PROGRAM MOTOR_FAULTS
VAR
	TON_GL1_MTR: TON; // MOTOR FAULT DELAY TIMER
	TON_GL2_MTR: TON; // MOTOR FAULT DELAY TIMER
	TON_GL3_MTR: TON; // MOTOR FAULT DELAY TIMER
	TON_GL4_MTR: TON; // MOTOR FAULT DELAY TIMER
	TON_GL5A_MTR: TON; // MOTOR FAULT DELAY TIMER
	TON_GL5B_MTR: TON; // MOTOR FAULT DELAY TIMER
	TON_GL6_MTR: TON; // MOTOR FAULT DELAY TIMER
	TON_GL7_MTR: TON; // MOTOR FAULT DELAY TIMER
	TON_GL8_MTR: TON; // MOTOR FAULT DELAY TIMER
	TON_GL9_MTR: TON; // MOTOR FAULT DELAY TIMER
	TON_GL10_MTR: TON; // MOTOR FAULT DELAY TIMER
	TON_GL11_MTR: TON; // MOTOR FAULT DELAY TIMER
	
	GL1_MTR: sClearPath;
	GL2_MTR: sClearPath;
	GL3_MTR: sClearPath;
	GL4_MTR: sClearPath;
	GL5_MTR: sClearPath;
	GL6_MTR: sClearPath;
	GL7_MTR: sClearPath;
	GL8_MTR: sClearPath;
	GL9_MTR: sClearPath;
	GL10_MTR: sClearPath;
	GL11_MTR: sClearPath;
		
	
	GL1: sTransfer;
	GL2: sTransfer;
	GL3: sConveyor;
	GL4: sConveyor;
	GL5A: sConveyor;
	GL5B: sConveyor;
	GL6: sConveyor;
	GL7:sConveyor;
	GL8: sConveyor;
	GL9: sConveyor;
	GL10: sConveyor;
	GL11: sConveyor;
	GL1_RD: SRoll_Door;
	

	RUN_FWD_TO_GL6_BIT : BOOL; // GL2 OCCUPIED, GL6 REQUESTING PART, RUN TO GL6 POSITION
	RUN_FWD_TO_GL8_BIT : BOOL; // GL2 OCCUPIED, GL8 REQUESTING PART, RUN TO GL8 POSITION
	RUN_REV_TO_GL5B_BIT : BOOL; //GL2 EMPTY, GL2 REQUESTING PART, RUN TO GL5 POSITION
	MTR_FAULT_PRESET_TIME: TIME; // FAULT TIMER PRESET TO MOTOR FAULT. DEFAULT IS 1000mS.
	COUNTER_PRESET: WORD; // MAX COUNT VALUE
	
	
END_VAR
VAR // added by the converter: edge detectors and wires of the graphical bodies
    _w1 : BOOL;
END_VAR

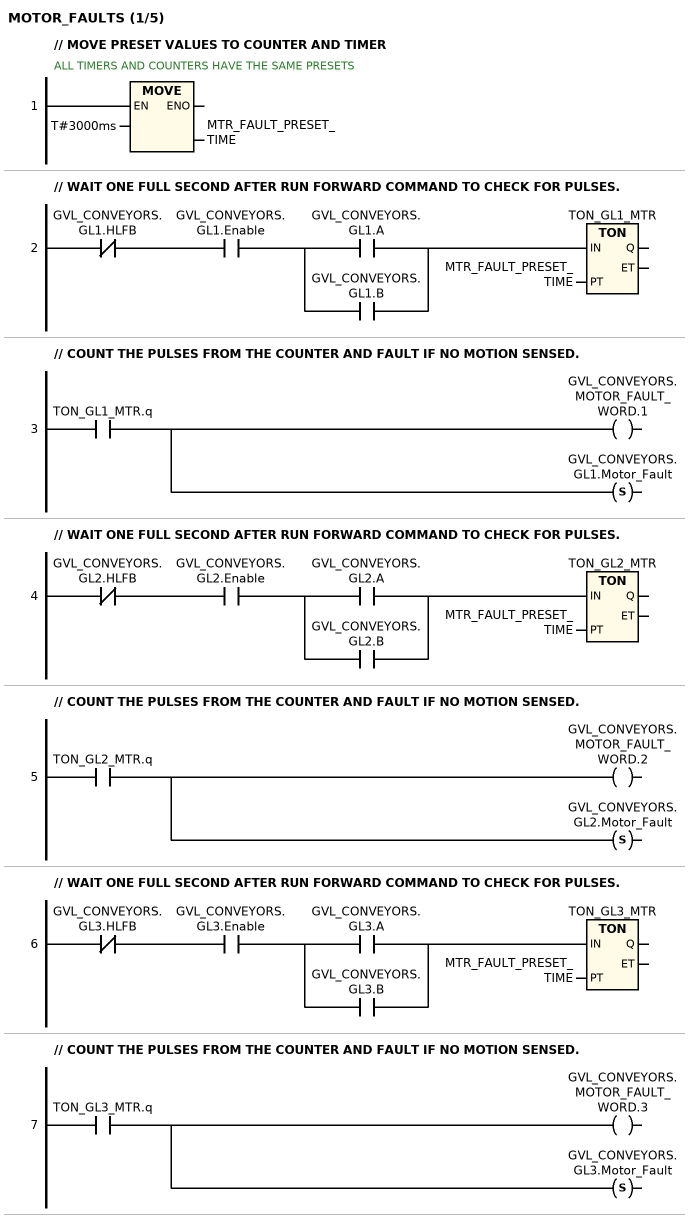
// NETWORK 1: // MOVE PRESET VALUES TO COUNTER AND TIMER
// ALL TIMERS AND COUNTERS HAVE THE SAME PRESETS
MTR_FAULT_PRESET_TIME := T#3000ms;

// NETWORK 2: // WAIT ONE FULL SECOND AFTER RUN FORWARD COMMAND TO CHECK FOR PULSES.
TON_GL1_MTR(IN := NOT GVL_CONVEYORS.GL1.HLFB AND GVL_CONVEYORS.GL1.Enable AND (GVL_CONVEYORS.GL1.A OR GVL_CONVEYORS.GL1.B), PT := MTR_FAULT_PRESET_TIME); // TON

// NETWORK 3: // COUNT THE PULSES FROM THE COUNTER AND FAULT IF NO MOTION SENSED.
GVL_CONVEYORS.MOTOR_FAULT_WORD.1 := TON_GL1_MTR.q;
GVL_CONVEYORS.GL1.Motor_Fault S= TON_GL1_MTR.q;

// NETWORK 4: // WAIT ONE FULL SECOND AFTER RUN FORWARD COMMAND TO CHECK FOR PULSES.
TON_GL2_MTR(IN := NOT GVL_CONVEYORS.GL2.HLFB AND GVL_CONVEYORS.GL2.Enable AND (GVL_CONVEYORS.GL2.A OR GVL_CONVEYORS.GL2.B), PT := MTR_FAULT_PRESET_TIME); // TON

// NETWORK 5: // COUNT THE PULSES FROM THE COUNTER AND FAULT IF NO MOTION SENSED.
GVL_CONVEYORS.MOTOR_FAULT_WORD.2 := TON_GL2_MTR.q;
GVL_CONVEYORS.GL2.Motor_Fault S= TON_GL2_MTR.q;

// NETWORK 6: // WAIT ONE FULL SECOND AFTER RUN FORWARD COMMAND TO CHECK FOR PULSES.
TON_GL3_MTR(IN := NOT GVL_CONVEYORS.GL3.HLFB AND GVL_CONVEYORS.GL3.Enable AND (GVL_CONVEYORS.GL3.A OR GVL_CONVEYORS.GL3.B), PT := MTR_FAULT_PRESET_TIME); // TON

// NETWORK 7: // COUNT THE PULSES FROM THE COUNTER AND FAULT IF NO MOTION SENSED.
GVL_CONVEYORS.MOTOR_FAULT_WORD.3 := TON_GL3_MTR.q;
GVL_CONVEYORS.GL3.Motor_Fault S= TON_GL3_MTR.q;

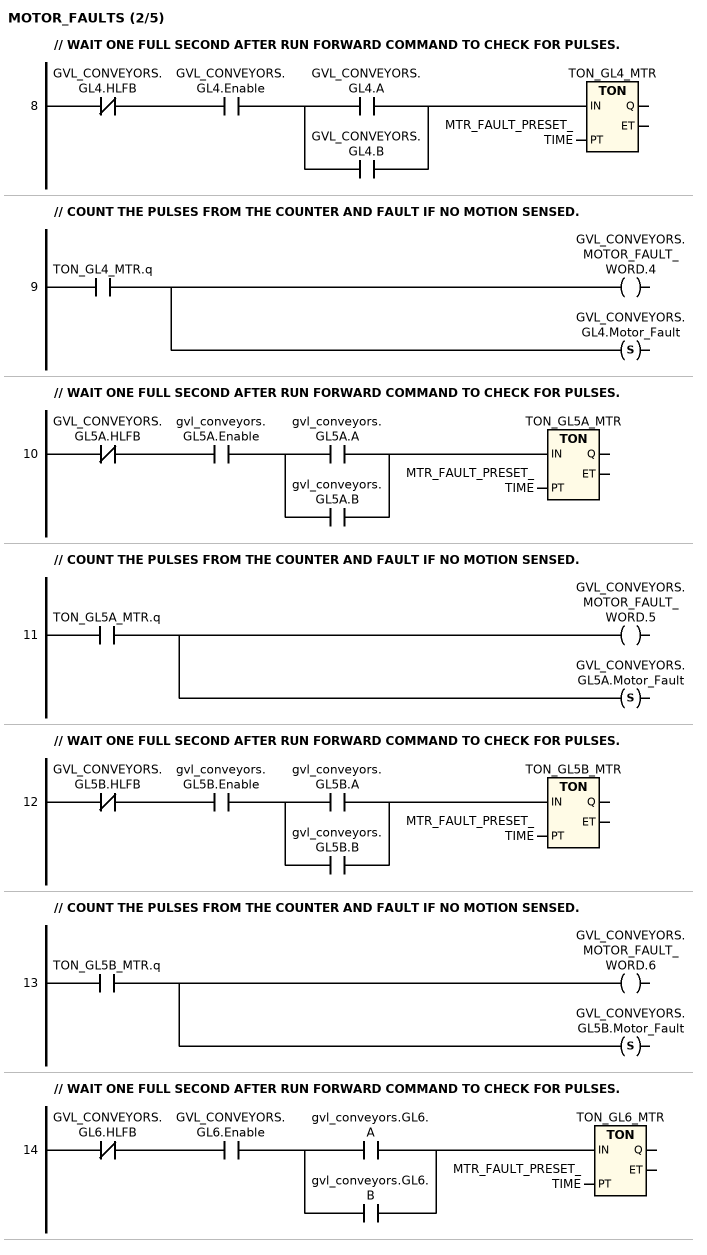
// NETWORK 8: // WAIT ONE FULL SECOND AFTER RUN FORWARD COMMAND TO CHECK FOR PULSES.
TON_GL4_MTR(IN := NOT GVL_CONVEYORS.GL4.HLFB AND GVL_CONVEYORS.GL4.Enable AND (GVL_CONVEYORS.GL4.A OR GVL_CONVEYORS.GL4.B), PT := MTR_FAULT_PRESET_TIME); // TON

// NETWORK 9: // COUNT THE PULSES FROM THE COUNTER AND FAULT IF NO MOTION SENSED.
GVL_CONVEYORS.MOTOR_FAULT_WORD.4 := TON_GL4_MTR.q;
GVL_CONVEYORS.GL4.Motor_Fault S= TON_GL4_MTR.q;

// NETWORK 10: // WAIT ONE FULL SECOND AFTER RUN FORWARD COMMAND TO CHECK FOR PULSES.
TON_GL5A_MTR(IN := NOT GVL_CONVEYORS.GL5A.HLFB AND gvl_conveyors.GL5A.Enable AND (gvl_conveyors.GL5A.A OR gvl_conveyors.GL5A.B), PT := MTR_FAULT_PRESET_TIME); // TON

// NETWORK 11: // COUNT THE PULSES FROM THE COUNTER AND FAULT IF NO MOTION SENSED.
GVL_CONVEYORS.MOTOR_FAULT_WORD.5 := TON_GL5A_MTR.q;
GVL_CONVEYORS.GL5A.Motor_Fault S= TON_GL5A_MTR.q;

// NETWORK 12: // WAIT ONE FULL SECOND AFTER RUN FORWARD COMMAND TO CHECK FOR PULSES.
TON_GL5B_MTR(IN := NOT GVL_CONVEYORS.GL5B.HLFB AND gvl_conveyors.GL5B.Enable AND (gvl_conveyors.GL5B.A OR gvl_conveyors.GL5B.B), PT := MTR_FAULT_PRESET_TIME); // TON

// NETWORK 13: // COUNT THE PULSES FROM THE COUNTER AND FAULT IF NO MOTION SENSED.
GVL_CONVEYORS.MOTOR_FAULT_WORD.6 := TON_GL5B_MTR.q;
GVL_CONVEYORS.GL5B.Motor_Fault S= TON_GL5B_MTR.q;

// NETWORK 14: // WAIT ONE FULL SECOND AFTER RUN FORWARD COMMAND TO CHECK FOR PULSES.
TON_GL6_MTR(IN := NOT GVL_CONVEYORS.GL6.HLFB AND GVL_CONVEYORS.GL6.Enable AND (gvl_conveyors.GL6.A OR gvl_conveyors.GL6.B), PT := MTR_FAULT_PRESET_TIME); // TON

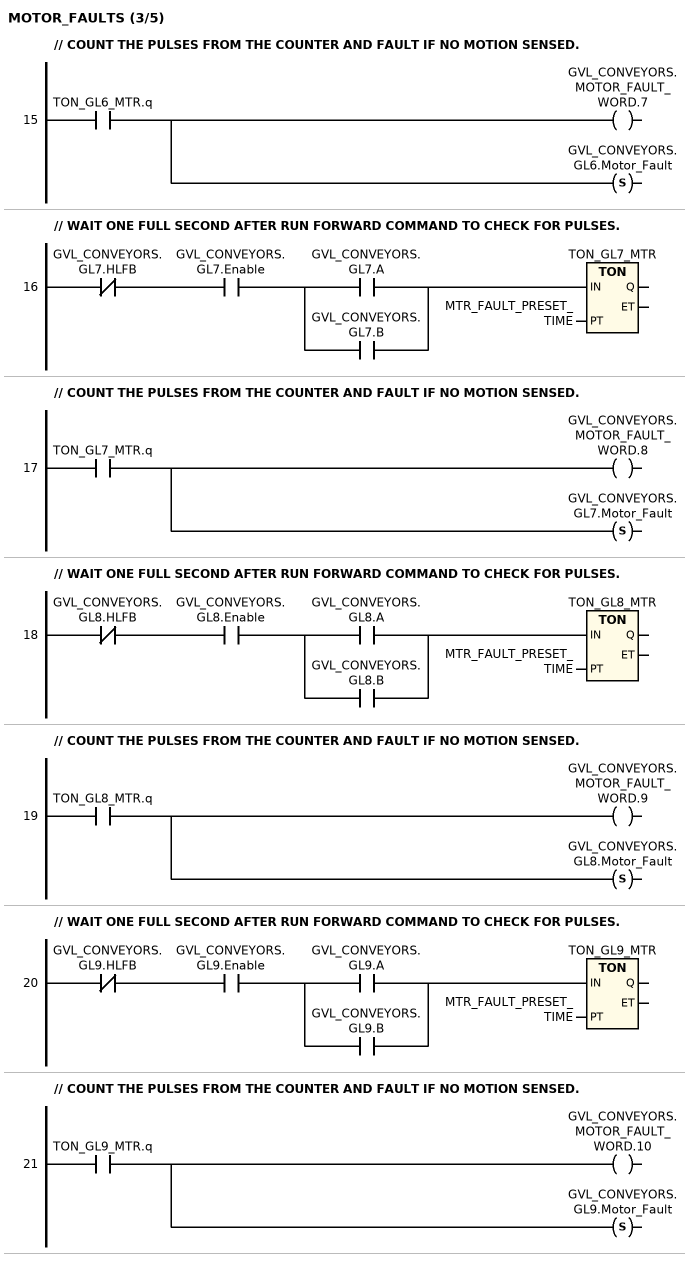
// NETWORK 15: // COUNT THE PULSES FROM THE COUNTER AND FAULT IF NO MOTION SENSED.
GVL_CONVEYORS.MOTOR_FAULT_WORD.7 := TON_GL6_MTR.q;
GVL_CONVEYORS.GL6.Motor_Fault S= TON_GL6_MTR.q;

// NETWORK 16: // WAIT ONE FULL SECOND AFTER RUN FORWARD COMMAND TO CHECK FOR PULSES.
TON_GL7_MTR(IN := NOT GVL_CONVEYORS.GL7.HLFB AND GVL_CONVEYORS.GL7.Enable AND (GVL_CONVEYORS.GL7.A OR GVL_CONVEYORS.GL7.B), PT := MTR_FAULT_PRESET_TIME); // TON

// NETWORK 17: // COUNT THE PULSES FROM THE COUNTER AND FAULT IF NO MOTION SENSED.
GVL_CONVEYORS.MOTOR_FAULT_WORD.8 := TON_GL7_MTR.q;
GVL_CONVEYORS.GL7.Motor_Fault S= TON_GL7_MTR.q;

// NETWORK 18: // WAIT ONE FULL SECOND AFTER RUN FORWARD COMMAND TO CHECK FOR PULSES.
TON_GL8_MTR(IN := NOT GVL_CONVEYORS.GL8.HLFB AND GVL_CONVEYORS.GL8.Enable AND (GVL_CONVEYORS.GL8.A OR GVL_CONVEYORS.GL8.B), PT := MTR_FAULT_PRESET_TIME); // TON

// NETWORK 19: // COUNT THE PULSES FROM THE COUNTER AND FAULT IF NO MOTION SENSED.
GVL_CONVEYORS.MOTOR_FAULT_WORD.9 := TON_GL8_MTR.q;
GVL_CONVEYORS.GL8.Motor_Fault S= TON_GL8_MTR.q;

// NETWORK 20: // WAIT ONE FULL SECOND AFTER RUN FORWARD COMMAND TO CHECK FOR PULSES.
TON_GL9_MTR(IN := NOT GVL_CONVEYORS.GL9.HLFB AND GVL_CONVEYORS.GL9.Enable AND (GVL_CONVEYORS.GL9.A OR GVL_CONVEYORS.GL9.B), PT := MTR_FAULT_PRESET_TIME); // TON

// NETWORK 21: // COUNT THE PULSES FROM THE COUNTER AND FAULT IF NO MOTION SENSED.
GVL_CONVEYORS.MOTOR_FAULT_WORD.10 := TON_GL9_MTR.q;
GVL_CONVEYORS.GL9.Motor_Fault S= TON_GL9_MTR.q;

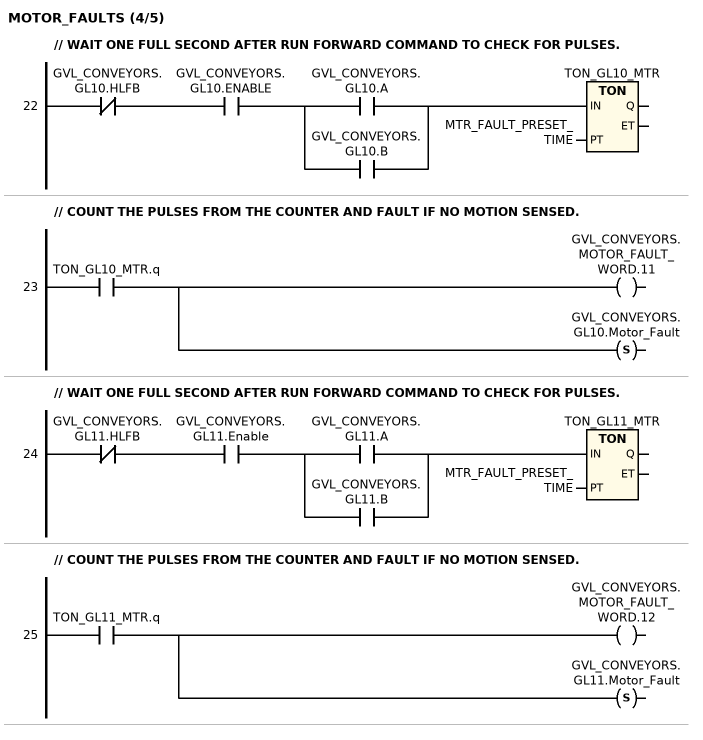
// NETWORK 22: // WAIT ONE FULL SECOND AFTER RUN FORWARD COMMAND TO CHECK FOR PULSES.
TON_GL10_MTR(IN := NOT GVL_CONVEYORS.GL10.HLFB AND GVL_CONVEYORS.GL10.ENABLE AND (GVL_CONVEYORS.GL10.A OR GVL_CONVEYORS.GL10.B), PT := MTR_FAULT_PRESET_TIME); // TON

// NETWORK 23: // COUNT THE PULSES FROM THE COUNTER AND FAULT IF NO MOTION SENSED.
GVL_CONVEYORS.MOTOR_FAULT_WORD.11 := TON_GL10_MTR.q;
GVL_CONVEYORS.GL10.Motor_Fault S= TON_GL10_MTR.q;

// NETWORK 24: // WAIT ONE FULL SECOND AFTER RUN FORWARD COMMAND TO CHECK FOR PULSES.
TON_GL11_MTR(IN := NOT GVL_CONVEYORS.GL11.HLFB AND GVL_CONVEYORS.GL11.Enable AND (GVL_CONVEYORS.GL11.A OR GVL_CONVEYORS.GL11.B), PT := MTR_FAULT_PRESET_TIME); // TON

// NETWORK 25: // COUNT THE PULSES FROM THE COUNTER AND FAULT IF NO MOTION SENSED.
GVL_CONVEYORS.MOTOR_FAULT_WORD.12 := TON_GL11_MTR.q;
GVL_CONVEYORS.GL11.Motor_Fault S= TON_GL11_MTR.q;

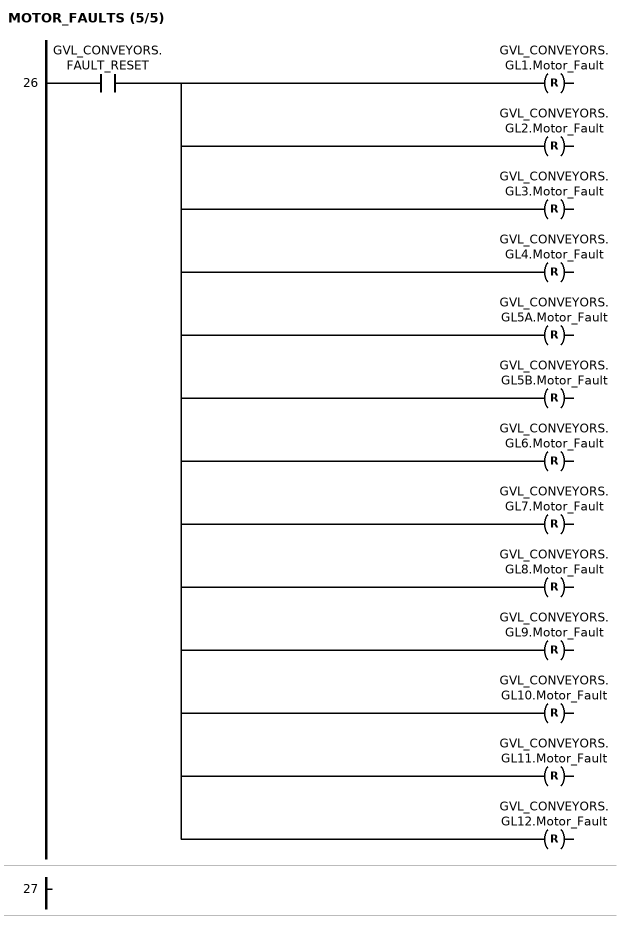
// NETWORK 26
_w1 := GVL_CONVEYORS.FAULT_RESET;
GVL_CONVEYORS.GL1.Motor_Fault R= _w1;
GVL_CONVEYORS.GL2.Motor_Fault R= _w1;
GVL_CONVEYORS.GL3.Motor_Fault R= _w1;
GVL_CONVEYORS.GL4.Motor_Fault R= _w1;
GVL_CONVEYORS.GL5A.Motor_Fault R= _w1;
GVL_CONVEYORS.GL5B.Motor_Fault R= _w1;
GVL_CONVEYORS.GL6.Motor_Fault R= _w1;
GVL_CONVEYORS.GL7.Motor_Fault R= _w1;
GVL_CONVEYORS.GL8.Motor_Fault R= _w1;
GVL_CONVEYORS.GL9.Motor_Fault R= _w1;
GVL_CONVEYORS.GL10.Motor_Fault R= _w1;
GVL_CONVEYORS.GL11.Motor_Fault R= _w1;
GVL_CONVEYORS.GL12.Motor_Fault R= _w1;

// NETWORK 27

END_PROGRAM

(* stored: Version 1.1.0.1, ProductVersion 3.1.4024.12
   POU MOTOR_FAULTS: Id {8267263e-a074-4a13-bf11-bbb79910f227}, SpecialFunc None *)
